{attribute 'qualified_only'}
VAR_GLOBAL PERSISTENT
	Tags: AdsTagsSmokeControl;
END_VAR

(* stored: Version 1.1.0.1, ProductVersion 3.1.4024.6
   GVL ADS_SmokeControl: Id {8f9ce8e0-d99d-4108-9603-3c79ea91e7cc} *)
